{attribute 'qualified_only'}
{attribute 'strict'}
TYPE E_States :
(
	Call := 0,
	MoveUp,
	MoveDown,
	SlowDown,
	Stop
);
END_TYPE

(* stored: Version 1.1.0.1, ProductVersion 3.1.4024.11
   DUT E_States: Id {df00cce3-a78a-4865-b4f7-28d0deec4f66} *)
